Staubli VAL3: chkDrivesOpEnab.pgx

program chkDrivesOpEnab()
  local num l_i
begin
  //检查驱动器是否使能
  bDrivesOpEnable=true
  for l_i=0 to nAxesSum-1
    if  nDrvState[l_i]==5
      bOpeEnabled[l_i]=true
    else
      bOpeEnabled[l_i]=false
    endIf
    bDrivesOpEnable=bDrivesOpEnable and  bOpeEnabled[l_i]
  endFor

//
//  bDrivesOpEnable=bOpeEnabled[0]=(diOpeEnabled[0]==true and diSwitchedOn[0]==true and diQuickStop[0]==true )
//  for l_i=1 to nAxesSum-1
//    bOpeEnabled[l_i]=(diOpeEnabled[l_i]==true and diQuickStop[l_i]==true and  diSwitchedOn[l_i]==true )
//   // bOpeEnabled[l_i]=(diOpeEnabled[0]==true  and  diSwitchedOn[0]==true )
//    bDrivesOpEnable=bDrivesOpEnable and bOpeEnabled[l_i]
//  endFor
end
